FUNCTION SCALE (* Scaling Function Block *)
  (* Standard: 61499-1; Description: Copyright (c) 2024 HR Agrartechnik GmbH This program and the accompanying materials are made available under the terms of the Eclipse Public License 2.0 which is available at https://www.eclipse.org/legal/epl-2.0/ SPDX-License-Identifier: EPL-2.0 was inspired by this Video: EP2 - CODESYS: Create Scaling Function Block https://www.youtube.com/watch?v=Ir6QAxxDarI *)
  (* Version 3.0, 2025-04-14, Patrick Aigner, changed package *)
  (* Version 1.0, 2024-09-19, Franz Höpfinger, HR Agrartechnik GmbH *)
  PACKAGE signalprocessing;
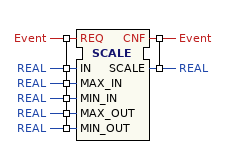
  EVENT_INPUT
    REQ WITH IN, MAX_IN, MIN_IN, MAX_OUT, MIN_OUT;
  END_EVENT
  EVENT_OUTPUT
    CNF WITH SCALE;
  END_EVENT
  VAR_INPUT
    IN : REAL; (* Input to be Scaled *)
    MAX_IN : REAL; (* Maximum Input *)
    MIN_IN : REAL; (* Minimum Input *)
    MAX_OUT : REAL; (* Maximum Ouput *)
    MIN_OUT : REAL; (* Minimum Output *)
  END_VAR
  VAR_OUTPUT
    SCALE : REAL;
  END_VAR
  BODY IN ST:
PACKAGE signalprocessing;

(* Scaling Function Block *)
FUNCTION SCALE : REAL
VAR_INPUT
	IN : REAL; // Input to be Scaled
	MAX_IN : REAL; // Maximum Input
	MIN_IN : REAL; // Minimum Input
	MAX_OUT : REAL; // Maximum Ouput
	MIN_OUT : REAL; // Minimum Output
END_VAR

SCALE := (IN - MIN_IN) * (MAX_OUT - MIN_OUT) / (MAX_IN - MIN_IN) + MIN_OUT;

END_FUNCTION
  END_BODY
END_FUNCTION
